TYPE ST_SM_StepInfo :
STRUCT
    CurrentStep : DINT;
    CurrentStepName : STRING(40);
    NextStep : DINT;
    StepTimerSeconds : REAL;
END_STRUCT
END_TYPE

(* stored: Version 1.1.0.1, ProductVersion 3.1.4024.13
   DUT ST_SM_StepInfo: Id {2cc141ff-dea0-456e-b495-38729cf383eb} *)
